Yaskawa INFORM job: X2_102(P)(90,-90)1.JBI

/JOB
//NAME X2_102(P)(90,-90)1
//POS
///NPOS 230,230,226,13,0,0
///TOOL 0
///POSTYPE PULSE
///PULSE
C00000=2000,-138093,-117084,0,0,0
C00001=4305,236497,208118,-17761,33698,0
C00002=-59706,236497,171970,-17761,33698,0
C00003=-68642,233553,162335,18407,63943,-60167
C00004=-68620,237873,184689,20710,53031,-62187
C00005=-67493,232083,179997,20020,52672,-61765
C00006=-67050,229604,177876,19730,52595,-61585
C00007=-67044,229502,178985,19916,51901,-61724
C00008=-67038,229450,178497,19841,52157,-61669
C00009=-66578,226776,174924,19337,52827,-61332
C00010=-67038,229450,178497,19841,52157,-61669
C00011=-68631,234094,163892,18504,63294,-60271
C00012=-68145,241811,194493,16574,45015,-61509
C00013=-67317,229778,184749,15987,44670,-61166
C00014=-67317,229387,185455,16165,44058,-61279
C00015=-67317,229778,184749,15987,44670,-61166
C00016=-66834,227293,181425,15407,45318,-60815
C00017=-67317,229778,184749,15987,44670,-61166
C00018=-68701,238087,188501,16512,46831,-61441
C00019=-66679,248207,214141,19957,35663,-62952
C00020=-66362,236944,211229,20590,32234,-63605
C00021=-65277,231220,208227,19566,31083,-63125
C00022=-65277,230538,208245,19768,30741,-63230
C00023=-65277,231220,208227,19566,31083,-63125
C00024=-64770,229332,205657,18720,31545,-62649
C00025=-65277,231220,208227,19566,31083,-63125
C00026=-63899,247748,213566,15829,35762,-61053
C00027=-132961,256009,219351,-662,67771,16322
C00028=-150721,258133,220838,-4903,56597,36219
C00029=-175956,234235,210676,-21015,30395,63926
C00030=-177622,226369,202159,-18586,31129,62559
C00031=-177622,225563,202167,-18810,30730,62676
C00032=-177622,225876,202166,-18723,30883,62631
C00033=-178207,223412,198783,-17689,31531,62057
C00034=-177236,228737,204255,-19030,31146,62814
C00035=-175884,240118,209836,-19152,33747,62947
C00036=-173679,229857,186287,-16925,43983,61731
C00037=-173679,227981,188546,-17672,41731,62191
C00038=-173679,227243,189165,-17934,41006,62348
C00039=-173679,227551,188921,-17828,41299,62281
C00040=-174254,224827,185246,-17073,41999,61834
C00041=-173679,227551,188921,-17828,41299,62281
C00042=-173139,236491,197187,-18441,40951,62645
C00043=-172603,232602,161257,-18712,64089,60261
C00044=-173924,235628,180815,-18889,51873,61342
C00045=-172608,237232,184033,-21073,53108,62337
C00046=-173740,231415,179286,-20377,52761,61910
C00047=-174186,228920,177136,-20083,52691,61728
C00048=-174192,228817,178244,-20271,51998,61869
C00049=-174189,228638,177277,-20141,52472,61772
C00050=-174651,225918,173635,-19633,53157,61430
C00051=-174189,228638,177277,-20141,52472,61772
C00052=-172611,236980,184222,-21136,52878,62385
C00053=-172606,232705,161920,-18764,63751,60317
C00054=-33909,232602,161257,-18712,64089,60261
C00055=-15700,2243,-58558,-65367,94407,-58645
C00056=-42038,-24148,-64629,-54323,75559,-58717
C00057=-44197,-22959,-60659,-53735,73332,-58425
C00058=-45039,-22397,-59015,-53526,72451,-58312
C00059=-44979,-23271,-57928,-53825,71802,-57871
C00060=-44992,-23122,-58143,-53767,71922,-57954
C00061=-46191,-21439,-56856,-53216,71335,-58219
C00062=-44992,-23122,-58143,-53767,71922,-57954
C00063=-41989,-25009,-63827,-54529,75024,-58350
C00064=-32524,-34812,-71854,-58522,80038,-56653
C00065=-45017,-81581,-97017,-55472,68259,-55558
C00066=-56084,-63511,-88405,-49217,64831,-59493
C00067=-58462,-60349,-83704,-48479,62782,-59568
C00068=-59376,-59036,-81788,-48205,61981,-59596
C00069=-59311,-59777,-80503,-48699,61221,-59131
C00070=-59003,-60257,-81034,-48822,61431,-59087
C00071=-60302,-57702,-79583,-47994,61058,-59566
C00072=-59003,-60257,-81034,-48822,61431,-59087
C00073=-55681,-64881,-87691,-49815,64278,-58966
C00074=-45017,-81581,-97017,-55472,68259,-55558
C00075=-32894,-34432,-71630,-58366,79867,-56737
C00076=-41688,-24576,-64954,-54484,75728,-58645
C00077=-43859,-23403,-60999,-53891,73497,-58353
C00078=-44706,-22847,-59360,-53679,72615,-58240
C00079=-44645,-23721,-58271,-53976,71967,-57798
C00080=-44682,-23582,-58448,-53916,72056,-57875
C00081=-45888,-21907,-57169,-53364,71466,-58140
C00082=-44682,-23582,-58448,-53916,72056,-57875
C00083=-41663,-25454,-64115,-54683,75164,-58270
C00084=-32894,-34432,-71630,-58366,79867,-56737
C00085=-30502,-36607,-73062,-59339,81056,-56251
C00086=-41630,-24614,-65007,-54508,75766,-58639
C00087=-43802,-23446,-61055,-53913,73534,-58347
C00088=-44650,-22892,-59418,-53701,72651,-58234
C00089=-44589,-23766,-58329,-53998,72004,-57792
C00090=-44608,-23720,-58520,-53955,72080,-57850
C00091=-45815,-22046,-57244,-53403,71488,-58116
C00092=-44608,-23720,-58520,-53955,72080,-57850
C00093=-41584,-25591,-64184,-54723,75189,-58245
C00094=-30502,-36607,-73062,-59339,81056,-56251
C00095=-30521,-36804,-72907,-59354,80942,-56176
C00096=-41810,-24598,-64713,-54460,75569,-58606
C00097=-43977,-23401,-60743,-53873,73340,-58316
C00098=-44823,-22836,-59099,-53664,72459,-58203
C00099=-44777,-23490,-58282,-53888,71973,-57872
C00100=-44767,-23386,-58412,-53859,72059,-57922
C00101=-45672,-22131,-57454,-53445,71616,-58121
C00102=-44767,-23386,-58412,-53859,72059,-57922
C00103=-41752,-25252,-64079,-54627,75166,-58318
C00104=-30521,-36804,-72907,-59354,80942,-56176
C00105=-48617,-100899,-104901,-55908,63245,-54221
C00106=-60981,-78178,-95502,-47940,60221,-59456
C00107=-63421,-73970,-90529,-47045,58377,-59730
C00108=-64353,-72276,-88515,-46711,57655,-59831
C00109=-64286,-72889,-87139,-47282,56881,-59359
C00110=-64274,-72850,-87331,-47224,56982,-59410
C00111=-65583,-69919,-85834,-46243,56736,-59988
C00112=-64274,-72850,-87331,-47224,56982,-59410
C00113=-57432,-98051,-106862,-51065,59935,-57313
C00114=-51188,-107076,-112538,-52509,60337,-56355
C00115=-83162,-143293,-113239,4095,19388,-67719
C00116=-87059,-126422,-104497,10100,20417,-69023
C00117=-85148,-116277,-98792,5838,21915,-66988
C00118=-84341,-113269,-97174,4239,22413,-66225
C00119=-41354,-51421,-69594,-68729,84300,-42170
C00120=-66411,-100108,-97884,-57632,66468,-44476
C00121=-56302,-60377,-70344,-75389,89529,-53167
C00122=-54473,-59290,-70505,-75710,90966,-53293
C00123=-50946,-58104,-72389,-76445,93850,-53772
C00124=-34731,-98541,-90949,-75868,93293,-49305
C00125=-38562,-61143,-74059,-78354,102200,-52510
C00126=-51313,-57535,-72089,-76390,93628,-53853
C00127=-54828,-58696,-70195,-75657,90754,-53377
C00128=-56440,-59997,-70035,-75367,89439,-53183
C00129=-93781,-139674,-106819,-38352,21241,-56382
C00130=-61530,-99076,-95664,-44966,45788,-52630
C00131=-83648,-111417,-96267,2924,22775,-65596
C00132=-85460,-115209,-98453,6324,22277,-67219
C00133=-87376,-128198,-110756,9444,23354,-68706
C00134=-66110,-162513,-113557,-65322,17781,-32754
C00135=-60362,-179762,-121914,-78103,19027,-26385
C00136=-78271,-141405,-108666,-10042,15201,-59438
C00137=-76792,-129799,-102924,-12030,17790,-58472
C00138=-74738,-129134,-99045,-25052,13652,-53297
C00139=-36188,-62041,-77688,-66032,84757,-42278
C00140=-46102,-88609,-90371,-65502,79628,-40662
C00141=-43207,-58645,-71334,-74593,95184,-49845
C00142=-41791,-47729,-64018,-78026,100149,-53095
C00143=-38644,-45375,-65147,-79031,102736,-53739
C00144=-22542,-58930,-72906,-80701,113358,-51531
C00145=-45507,-85827,-81768,-80030,94289,-48289
C00146=-21007,-49469,-63567,-84664,112915,-50403
C00147=-24143,-52779,-63157,-83372,110435,-49576
C00148=-25588,-55109,-63516,-82813,109262,-49172
C00149=-29213,-141193,-106326,-70590,66679,-33929
C00150=-21677,-102038,-94363,-66600,73853,-38839
C00151=-30241,-129324,-100953,-69122,50791,-33041
C00152=-46232,-152372,-104130,-83256,26044,-24905
C00153=-44377,-165065,-109179,-90053,27028,-21315
C00154=-311,-178979,-111450,-86459,56764,-16230
C00155=-59708,-176831,-116235,-83669,15342,-24345
C00156=-79056,-141883,-108790,-8064,14946,-60379
C00157=-77513,-130262,-103056,-10505,17536,-59201
C00158=-74170,-126151,-101228,-19436,19691,-55187
C00159=-36840,-62408,-78088,-65333,83828,-45019
C00160=-50437,-100078,-97430,-60201,71072,-46441
C00161=-45392,-83282,-85893,-68940,82387,-50193
C00162=-37649,-79344,-88446,-70118,88865,-50776
C00163=-26650,-88423,-96706,-71980,96311,-49687
C00164=-27360,-157090,-119697,-70425,73735,-40403
C00165=-26933,-67218,-77205,-79449,109983,-51051
C00166=-40780,-54413,-70384,-78301,100955,-53239
C00167=-44144,-56530,-69031,-77374,98185,-52627
C00168=-46739,-82554,-83925,-71442,84833,-50278
C00169=-64576,-133797,-108987,-56957,49971,-40299
C00170=-55730,-116486,-104453,-54149,57147,-39702
C00171=-64775,-126412,-104837,-43035,33616,-45207
C00172=-84360,-137825,-105111,6410,14710,-67243
C00173=-83782,-174049,-119465,14191,4988,-70704
C00174=4306,-189564,-118248,-76797,69073,-14089
C00175=-9355,229277,174760,14349,4120,-60080
C00176=-63851,249906,184838,11388,54090,-58270
C00177=-66966,229251,175893,14496,49590,-60184
C00178=-66966,228979,178450,14872,47930,-60442
C00179=-66981,229181,177726,14757,48464,-60364
C00180=-67823,233206,185230,16003,46159,-61141
C00181=-66981,228894,179384,15025,47334,-60544
C00182=-66990,228821,179287,15027,47357,-60545
C00183=-66967,228791,179403,15048,47276,-60547
C00184=-66961,228789,179266,15001,47362,-60537
C00185=-66965,228460,180628,15248,46388,-60700
C00186=-66802,227674,179068,14990,46895,-60538
C00187=-66779,227397,179466,15054,46528,-60590
C00188=-66807,226773,182027,15552,44699,-60914
C00189=-66832,224442,185298,16520,41608,-61494
C00190=-66840,224422,185215,16494,41648,-61489
C00191=-66820,223938,186111,16728,40875,-61637
C00192=-66853,222022,186802,17225,39537,-61929
C00193=-66912,216121,188235,18844,35797,-62842
C00194=-66885,216347,188464,18827,35771,-62831
C00195=-66952,215633,187924,18914,35747,-62874
C00196=-67008,215777,188020,18974,35761,-62903
C00197=-64896,228147,204946,18938,31412,-62768
C00198=-64451,229383,207615,19004,30362,-62779
C00199=-64319,229986,208437,18975,30146,-62755
C00200=-64320,235654,207860,17333,33259,-61891
C00201=-127852,233528,172858,-1116,53739,8677
C00202=-174263,228432,175140,-14901,49789,60445
C00203=-174268,228211,177769,-15284,48114,60710
C00204=-174246,228391,177829,-15287,48171,60710
C00205=-173475,232193,184234,-16357,46404,61376
C00206=-174246,228181,178891,-15468,47435,60832
C00207=-174240,228133,178826,-15469,47451,60832
C00208=-174271,228016,178845,-15463,47379,60831
C00209=-174276,227918,178508,-15413,47528,60799
C00210=-174286,227658,179844,-15655,46590,60950
C00211=-174351,227295,179377,-15579,46676,60907
C00212=-174332,227272,179929,-15676,46343,60972
C00213=-174371,226155,181833,-16121,44653,61258
C00214=-174192,224903,185875,-17238,41679,61934
C00215=-174186,224802,185663,-17218,41757,61925
C00216=-174205,224201,186288,-17427,41100,62055
C00217=-174226,222498,187148,-17913,39751,62341
C00218=-174338,216137,187971,-19375,36146,63177
C00219=-174344,216285,188030,-19351,36181,63161
C00220=-174327,216170,187871,-19349,36222,63161
C00221=-174333,215937,187942,-19432,36065,63204
C00222=-174325,215982,187948,-19443,36091,63210
C00223=-176900,230407,207583,-19326,31072,63020
C00224=-176902,229512,207806,-19651,30509,63187
C00225=-177018,230048,208538,-19629,30316,63168
C00226=-177017,235510,208022,-18011,33280,62316
C00227=-177018,208627,156143,-19629,29463,63168
C00228=4305,194232,136177,-17761,33698,62179
C00229=2000,-138093,-117084,0,0,0
BC00000=166720,666220,1057063
BC00001=32490,666220,1075175
BC00002=32490,666220,1075175
BC00003=108321,818406,1075175
BC00004=108321,818406,1075175
BC00005=108321,818406,1075175
BC00006=108321,818406,1075175
BC00007=108321,818406,1075175
BC00008=108321,818406,1075175
BC00009=108321,818406,1075175
BC00010=108321,818406,1075175
BC00011=108321,818406,1075175
BC00012=112515,736490,1075175
BC00013=112515,736490,1075175
BC00014=112515,736490,1075175
BC00015=112515,736490,1075175
BC00016=112515,736490,1075175
BC00017=112515,736490,1075175
BC00018=112515,736490,1075175
BC00019=112881,691782,1025034
BC00020=113047,671527,1002318
BC00021=113089,666372,996537
BC00022=113089,666372,996537
BC00023=113089,666372,996537
BC00024=113089,666372,996537
BC00025=113089,666372,996537
BC00026=113089,666372,996537
BC00027=249276,665500,992981
BC00028=284297,665276,992066
BC00029=334133,666220,990764
BC00030=334133,666220,990764
BC00031=334133,666220,990764
BC00032=334133,666220,990764
BC00033=334133,666220,990764
BC00034=334133,666220,990764
BC00035=334133,666220,990764
BC00036=325487,705237,1075175
BC00037=325487,705237,1075175
BC00038=325487,705237,1075175
BC00039=325487,705237,1075175
BC00040=325487,705237,1075175
BC00041=325487,705237,1075175
BC00042=325487,705237,1075175
BC00043=330094,817929,1075175
BC00044=331720,756851,1041191
BC00045=330094,817929,1075175
BC00046=330094,817929,1075175
BC00047=330094,817929,1075175
BC00048=330094,817929,1075175
BC00049=330094,817929,1075175
BC00050=330094,817929,1075175
BC00051=330094,817929,1075175
BC00052=330094,817929,1075175
BC00053=330094,817929,1075175
BC00054=52198,668359,1075175
BC00055=166720,666220,1057063
BC00056=216765,666220,1057063
BC00057=216765,666220,1057063
BC00058=216765,666220,1057063
BC00059=216765,666220,1057063
BC00060=216765,666220,1057063
BC00061=216765,666220,1057063
BC00062=216765,666220,1057063
BC00063=216765,666220,1057063
BC00064=216765,666220,1057063
BC00065=189956,666220,1056793
BC00066=189956,666220,1056793
BC00067=189956,666220,1056793
BC00068=189956,666220,1056793
BC00069=189956,666220,1056793
BC00070=189956,666220,1056793
BC00071=189956,666220,1056793
BC00072=189956,666220,1056793
BC00073=189956,666220,1056793
BC00074=189956,666220,1056793
BC00075=95589,666220,1056895
BC00076=95589,666220,1056895
BC00077=95589,666220,1056895
BC00078=95589,666220,1056895
BC00079=95589,666220,1056895
BC00080=95589,666220,1056895
BC00081=95589,666220,1056895
BC00082=95589,666220,1056895
BC00083=95589,666220,1056895
BC00084=95589,666220,1056895
BC00085=65057,666220,1056713
BC00086=65057,666220,1056713
BC00087=65057,666220,1056713
BC00088=65057,666220,1056713
BC00089=65057,666220,1056713
BC00090=65057,666220,1056713
BC00091=65057,666220,1056713
BC00092=65057,666220,1056713
BC00093=65057,666220,1056713
BC00094=65057,666220,1056713
BC00095=13150,666220,1055634
BC00096=13150,666220,1055634
BC00097=13150,666220,1055634
BC00098=13150,666220,1055634
BC00099=13150,666220,1055634
BC00100=13150,666220,1055634
BC00101=13150,666220,1055634
BC00102=13150,666220,1055634
BC00103=13150,666220,1055634
BC00104=13150,666220,1055634
BC00105=15,666220,1056645
BC00106=15,666220,1056645
BC00107=15,666220,1056645
BC00108=15,666220,1056645
BC00109=15,666220,1056645
BC00110=15,666220,1056645
BC00111=15,666220,1056645
BC00112=15,666220,1056645
BC00113=15,666220,1056645
BC00114=15,666220,1056645
BC00115=23745,686641,1073486
BC00116=26125,688689,1075175
BC00117=26125,688689,1075175
BC00118=26125,688689,1075175
BC00119=26125,688689,1075175
BC00120=26125,688689,1075175
BC00121=26125,688689,1075175
BC00122=26125,688689,1075175
BC00123=26125,688689,1075175
BC00124=26125,688689,1075175
BC00125=284154,689569,1075175
BC00126=284154,689569,1075175
BC00127=284154,689569,1075175
BC00128=284154,689569,1075175
BC00129=284154,689569,1075175
BC00130=284154,689569,1075175
BC00131=284154,689569,1075175
BC00132=284154,689569,1075175
BC00133=284154,689569,1075175
BC00134=284154,689569,1075175
BC00135=166821,701812,1075175
BC00136=166821,701812,1075175
BC00137=166821,701812,1075175
BC00138=166821,701812,1075175
BC00139=166821,701812,1075175
BC00140=166821,701812,1075175
BC00141=166821,701812,1075174
BC00142=166821,701812,1075175
BC00143=166821,701812,1075175
BC00144=166821,701812,1075175
BC00145=107577,675403,1075175
BC00146=60976,728964,1075175
BC00147=60976,728964,1075175
BC00148=60976,728964,1075175
BC00149=60976,728964,1075175
BC00150=60976,728964,1075175
BC00151=60975,728964,1075174
BC00152=60976,728964,1075175
BC00153=60976,728964,1075175
BC00154=60976,728964,1075175
BC00155=214157,701974,1075175
BC00156=214157,701974,1075175
BC00157=214157,701974,1075175
BC00158=214157,701974,1075175
BC00159=214157,701974,1075175
BC00160=214157,701974,1075175
BC00161=214157,701974,1075175
BC00162=214157,701974,1075175
BC00163=214157,701974,1075175
BC00164=214157,701974,1075175
BC00165=126731,702207,1075175
BC00166=126731,702207,1075175
BC00167=126731,702207,1075175
BC00168=126731,702207,1075175
BC00169=126731,702207,1075175
BC00170=126731,702207,1075175
BC00171=126731,702207,1075175
BC00172=126731,702207,1075175
BC00173=126731,702207,1075175
BC00174=126731,702207,1075175
BC00175=0,671300,1075175
BC00176=102033,814443,1075175
BC00177=104277,804739,1075175
BC00178=109889,805427,1075175
BC00179=112133,805702,1075175
BC00180=112133,805702,1075175
BC00181=112133,805702,1075175
BC00182=112133,805702,1075175
BC00183=112115,811337,1075171
BC00184=112235,790267,1075175
BC00185=112385,757219,1075175
BC00186=112368,762877,1075175
BC00187=112401,759711,1075175
BC00188=112515,736490,1075175
BC00189=112651,705808,1075172
BC00190=112632,711465,1075175
BC00191=112664,708917,1075175
BC00192=112731,698583,1075175
BC00193=112912,671578,1075175
BC00194=112897,675330,1075175
BC00195=112903,675530,1064805
BC00196=112969,667577,1038313
BC00197=113089,666372,996537
BC00198=110434,666220,999205
BC00199=104822,666220,1018123
BC00200=104780,666220,1075175
BC00201=236932,745843,1075175
BC00202=332819,804241,1075175
BC00203=327209,804894,1075175
BC00204=324965,805156,1075175
BC00205=324965,805156,1075175
BC00206=324965,805156,1075175
BC00207=324965,805156,1075175
BC00208=324947,810790,1075175
BC00209=325043,789742,1075175
BC00210=325218,756702,1075175
BC00211=325200,762360,1075175
BC00212=325209,759192,1075175
BC00213=325324,735955,1075175
BC00214=325487,705242,1075175
BC00215=325468,710849,1075175
BC00216=325473,708338,1075175
BC00217=325540,697985,1075175
BC00218=325697,671186,1075175
BC00219=325677,676538,1075175
BC00220=325677,676538,1075175
BC00221=325711,674865,1062596
BC00222=325783,666243,1034429
BC00223=325896,666237,989644
BC00224=328141,666220,997078
BC00225=333753,666220,1016016
BC00226=333712,666220,1075175
BC00227=333753,666220,1016016
BC00228=32490,666220,1075175
BC00229=166720,666220,1057063
EC00000=798156,-556475
EC00001=798156,-556920
EC00002=798156,-556920
EC00003=443420,-556475
EC00004=443420,-556475
EC00005=443420,-556475
EC00006=443420,-556475
EC00007=443420,-556475
EC00008=443420,-556475
EC00009=443420,-556475
EC00010=443420,-556475
EC00011=443420,-556475
EC00012=657016,-556187
EC00013=657016,-556187
EC00014=657016,-556187
EC00015=657016,-556187
EC00016=657016,-556187
EC00017=657016,-556187
EC00018=657016,-556187
EC00019=846901,-556371
EC00020=932929,-556454
EC00021=954822,-556475
EC00022=954822,-556475
EC00023=954822,-556475
EC00024=954822,-556475
EC00025=954822,-556475
EC00026=954822,-556475
EC00027=958275,-556749
EC00028=959163,-556820
EC00029=960426,-556920
EC00030=960426,-556920
EC00031=960426,-556920
EC00032=960426,-556920
EC00033=960426,-556920
EC00034=960426,-556920
EC00035=960426,-556920
EC00036=736908,-556362
EC00037=736908,-556362
EC00038=736908,-556362
EC00039=736908,-556362
EC00040=736908,-556362
EC00041=736908,-556362
EC00042=736908,-556362
EC00043=443420,-556475
EC00044=651568,-556654
EC00045=443420,-556475
EC00046=443420,-556475
EC00047=443420,-556475
EC00048=443420,-556475
EC00049=443420,-556475
EC00050=443420,-556475
EC00051=443420,-556475
EC00052=443420,-556475
EC00053=443420,-556475
EC00054=663289,-556475
EC00055=798156,-556475
EC00056=798156,-556475
EC00057=798156,-556475
EC00058=798156,-556475
EC00059=798156,-556475
EC00060=798156,-556475
EC00061=798156,-556475
EC00062=798156,-556475
EC00063=798156,-556475
EC00064=798156,-556475
EC00065=798156,-556475
EC00066=798156,-556475
EC00067=798156,-556475
EC00068=798156,-556475
EC00069=798156,-556475
EC00070=798156,-556475
EC00071=798156,-556475
EC00072=798156,-556475
EC00073=798156,-556475
EC00074=798156,-556475
EC00075=798156,-556475
EC00076=798156,-556475
EC00077=798156,-556475
EC00078=798156,-556475
EC00079=798156,-556475
EC00080=798156,-556475
EC00081=798156,-556475
EC00082=798156,-556475
EC00083=798156,-556475
EC00084=798156,-556475
EC00085=798156,-556475
EC00086=798156,-556475
EC00087=798156,-556475
EC00088=798156,-556475
EC00089=798156,-556475
EC00090=798156,-556475
EC00091=798156,-556475
EC00092=798156,-556475
EC00093=798156,-556475
EC00094=798156,-556475
EC00095=798156,-556475
EC00096=798156,-556475
EC00097=798156,-556475
EC00098=798156,-556475
EC00099=798156,-556475
EC00100=798156,-556475
EC00101=798156,-556475
EC00102=798156,-556475
EC00103=798156,-556475
EC00104=798156,-556475
EC00105=798156,-556475
EC00106=798156,-556475
EC00107=798156,-556475
EC00108=798156,-556475
EC00109=798156,-556475
EC00110=798156,-556475
EC00111=798156,-556475
EC00112=798156,-556475
EC00113=798156,-556475
EC00114=798156,-556475
EC00115=798156,-556475
EC00116=798156,-556475
EC00117=798156,-556475
EC00118=798156,-556475
EC00119=798156,-556475
EC00120=798156,-556475
EC00121=798156,-556475
EC00122=798156,-556475
EC00123=798156,-556475
EC00124=798156,-556475
EC00125=798156,-556475
EC00126=798156,-556475
EC00127=798156,-556475
EC00128=798156,-556475
EC00129=798156,-556475
EC00130=798156,-556475
EC00131=798156,-556475
EC00132=798156,-556475
EC00133=798156,-556475
EC00134=798156,-556475
EC00135=798156,-556475
EC00136=798156,-556475
EC00137=798156,-556475
EC00138=798156,-556475
EC00139=798156,-556475
EC00140=798156,-556475
EC00141=798155,-556475
EC00142=798156,-556475
EC00143=798156,-556475
EC00144=798156,-556475
EC00145=798156,-556475
EC00146=798156,-556475
EC00147=798156,-556475
EC00148=798156,-556475
EC00149=798156,-556475
EC00150=798156,-556475
EC00151=798155,-556475
EC00152=798156,-556475
EC00153=798156,-556475
EC00154=798156,-556475
EC00155=798156,-556475
EC00156=798156,-556475
EC00157=798156,-556475
EC00158=798156,-556475
EC00159=798156,-556475
EC00160=798156,-556475
EC00161=798156,-556475
EC00162=798156,-556475
EC00163=798156,-556475
EC00164=798156,-556475
EC00165=798156,-556475
EC00166=798156,-556475
EC00167=798156,-556475
EC00168=798156,-556475
EC00169=798156,-556475
EC00170=798156,-556475
EC00171=798156,-556475
EC00172=798156,-556475
EC00173=798156,-556475
EC00174=798156,-556475
EC00175=798156,-556475
EC00176=449706,-555609
EC00177=449706,-555609
EC00178=449706,-555609
EC00179=449706,-555609
EC00180=449706,-555609
EC00181=449704,-555609
EC00182=497563,-555770
EC00183=577410,-555996
EC00184=577410,-555996
EC00185=593464,-556037
EC00186=657016,-556187
EC00187=736906,-556362
EC00188=736908,-556362
EC00189=752993,-556395
EC00190=784818,-556475
EC00191=864675,-556475
EC00192=864752,-556475
EC00193=880165,-556475
EC00194=910304,-556475
EC00195=954822,-556475
EC00196=960426,-556475
EC00197=960426,-556475
EC00198=960426,-556475
EC00199=665239,-555975
EC00200=449706,-555609
EC00201=449706,-555609
EC00202=449706,-555609
EC00203=449706,-555609
EC00204=449706,-555609
EC00205=497563,-555770
EC00206=577410,-555996
EC00207=577410,-555996
EC00208=593464,-556037
EC00209=657016,-556187
EC00210=736908,-556362
EC00211=736908,-556362
EC00212=752993,-556395
EC00213=784818,-556475
EC00214=863892,-556660
EC00215=864791,-556662
EC00216=864791,-556662
EC00217=880786,-556704
EC00218=912696,-556789
EC00219=960272,-556920
EC00220=960426,-556920
EC00221=960426,-556920
EC00222=960426,-556920
EC00223=960426,-556920
EC00224=960426,-556920
EC00225=798156,-556475
///POSTYPE BASE
///RECTAN
///RCONF 0,0,0,0,0,0,0,0,0,0,0,0,0,0,0,0,0,0,0,0,0,0,0,0
P00006=0.222,-3.123,-1.508,0.0000,0.0000,0.0000
P00021=-0.225,-6.128,-0.405,0.0000,0.0000,0.0000
P00022=0.222,-3.123,-1.508,0.0000,0.0000,0.0000
P00023=0.143,-0.036,0.682,0.0000,0.0000,0.0000
P00024=0.145,-0.552,1.326,0.0000,0.0000,0.0000
P00025=-2.003,0.006,0.728,0.0000,0.0000,0.0000
P00026=0.562,-0.002,-0.337,0.0000,0.0000,0.0000
P00027=-0.746,0.015,-9.096,0.0000,0.0000,0.0000
P00028=-2.237,-0.018,-7.702,0.0000,0.0000,0.0000
P00066=5.557,-0.028,3.115,0.0000,0.0000,0.0000
///RCONF 0,1,0,0,0,0,0,0,0,0,0,0,0,0,0,0,0,0,0,0,0,0,0,0
P00067=-0.081,0.026,-1.119,0.0000,0.0000,0.0000
///RCONF 0,0,0,0,0,0,0,0,0,0,0,0,0,0,0,0,0,0,0,0,0,0,0,0
P00068=2.896,1.192,4.622,0.0000,0.0000,0.0000
///RCONF 0,1,0,0,0,0,0,0,0,0,0,0,0,0,0,0,0,0,0,0,0,0,0,0
P00075=-1.802,0.025,1.546,0.0000,0.0000,0.0000
//INST
///DATE 2024/04/10 12:22
///ATTR SC,RW
///GROUP1 RB1,BS1
///GROUP2 ST1
NOP
'X2_102(P)(90,-90)1
MOVJ C00000 BC00000 VJ=100.00  +MOVJ EC00000 VJ=100.00
MOVJ C00001 BC00001 VJ=100.00  +MOVJ EC00001 VJ=100.00
MOVJ C00002 BC00002 VJ=100.00  +MOVJ EC00002 VJ=100.00
'Path S3368
SFTOF3D
MOVJ C00003 BC00003 VJ=100.00  +MOVJ EC00003 VJ=100.00
MOVJ C00004 BC00004 VJ=100.00  +MOVJ EC00004 VJ=100.00
MOVL C00005 BC00005 V=800.0  +MOVJ EC00005 VJ=100.00
SMOVL C00006 BC00006 V=166.7  +MOVJ EC00006
SREFP 3 C00007 BC00007  +REFP EC00007
CALL JOB:SEARCH-R1-S13D
SET P027 P006
SFTON3D P027
SMOVL C00008 BC00008 V=166.7  +MOVJ EC00008
SREFP 3 C00009 BC00009  +REFP EC00009
CALL JOB:SEARCH-R1-S13D
SET P027 P006
SFTON3D P027
SMOVL C00010 BC00010 V=166.7  +MOVJ EC00010
MOVL C00011 BC00011 V=1000.0  +MOVJ EC00011 VJ=100.00
'EndPath S3368
'Path S3369
SFTOF3D
MOVJ C00012 BC00012 VJ=100.00  +MOVJ EC00012 VJ=100.00
SMOVL C00013 BC00013 V=250.0  +MOVJ EC00013
SREFP 3 C00014 BC00014  +REFP EC00014
CALL JOB:SEARCH-R1-S13D
SET P066 P006
SFTON3D P066
SMOVL C00015 BC00015 V=166.7  +MOVJ EC00015
SREFP 3 C00016 BC00016  +REFP EC00016
CALL JOB:SEARCH-R1-S13D
SET P066 P006
SFTON3D P066
SMOVL C00017 BC00017 V=250.0  +MOVJ EC00017
SFTOF3D
MOVJ C00018 BC00018 VJ=100.00  +MOVJ EC00018 VJ=100.00
MOVJ C00019 BC00019 VJ=100.00  +MOVJ EC00019 VJ=100.00
MOVJ C00020 BC00020 VJ=100.00  +MOVJ EC00020 VJ=100.00
SMOVL C00021 BC00021 V=250.0  +MOVJ EC00021
SREFP 3 C00022 BC00022  +REFP EC00022
CALL JOB:SEARCH-R1-S13D
SET P067 P006
SFTON3D P067
SMOVL C00023 BC00023 V=166.7  +MOVJ EC00023
SREFP 3 C00024 BC00024  +REFP EC00024
CALL JOB:SEARCH-R1-S13D
SET P067 P006
SFTON3D P067
SMOVL C00025 BC00025 V=250.0  +MOVJ EC00025
SFTOF3D
MOVJ C00026 BC00026 VJ=100.00  +MOVJ EC00026 VJ=100.00
MOVJ C00027 BC00027 VJ=40.00  +MOVJ EC00027 VJ=100.00
MOVJ C00028 BC00028 VJ=80.00  +MOVJ EC00028 VJ=100.00
SFTOF3D
MOVJ C00029 BC00029 VJ=80.00  +MOVJ EC00029 VJ=100.00
SMOVL C00030 BC00030 V=166.7  +MOVJ EC00030
SREFP 3 C00031 BC00031  +REFP EC00031
CALL JOB:SEARCH-R1-S13D
SET P068 P006
SFTON3D P068
SMOVL C00032 BC00032 V=166.7  +MOVJ EC00032
SREFP 3 C00033 BC00033  +REFP EC00033
CALL JOB:SEARCH-R1-S13D
SET P068 P006
SFTON3D P068
SMOVL C00034 BC00034 V=250.0  +MOVJ EC00034
SFTOF3D
MOVJ C00035 BC00035 VJ=80.00  +MOVJ EC00035 VJ=80.00
MOVJ C00036 BC00036 VJ=100.00  +MOVJ EC00036 VJ=100.00
SFTOF3D
SMOVL C00037 BC00037 V=166.7  +MOVJ EC00037
SREFP 3 C00038 BC00038  +REFP EC00038
CALL JOB:SEARCH-R1-S13D
SET P075 P006
SFTON3D P075
SMOVL C00039 BC00039 V=166.7  +MOVJ EC00039
SREFP 3 C00040 BC00040  +REFP EC00040
CALL JOB:SEARCH-R1-S13D
SET P075 P006
SFTON3D P075
SMOVL C00041 BC00041 V=250.0  +MOVJ EC00041
SFTOF3D
MOVL C00042 BC00042 V=1000.0  +MOVJ EC00042 VJ=100.00
MOVJ C00043 BC00043 VJ=100.00  +MOVJ EC00043 VJ=100.00
MOVJ C00044 BC00044 VJ=100.00  +MOVJ EC00044 VJ=100.00
MOVJ C00045 BC00045 VJ=100.00  +MOVJ EC00045 VJ=100.00
MOVL C00046 BC00046 V=800.0  +MOVJ EC00046 VJ=100.00
SMOVL C00047 BC00047 V=166.7  +MOVJ EC00047
SREFP 3 C00048 BC00048  +REFP EC00048
CALL JOB:SEARCH-R1-S13D
SET P028 P006
SFTON3D P028
SMOVL C00049 BC00049 V=166.7  +MOVJ EC00049
SREFP 3 C00050 BC00050  +REFP EC00050
CALL JOB:SEARCH-R1-S13D
SET P028 P006
SFTON3D P028
SMOVL C00051 BC00051 V=250.0  +MOVJ EC00051
MOVL C00052 BC00052 V=1000.0  +MOVJ EC00052 VJ=100.00
MOVL C00053 BC00053 V=1000.0  +MOVJ EC00053 VJ=100.00
'EndPath S3369
MOVJ C00054 BC00054 VJ=100.00  +MOVJ EC00054 VJ=100.00
'
MOVJ C00055 BC00055 VJ=100.00  +MOVJ EC00055 VJ=100.00
'Path S3399
SFTOF3D
MOVJ C00056 BC00056 VJ=100.00  +MOVJ EC00056 VJ=100.00
MOVL C00057 BC00057 V=800.0  +MOVJ EC00057 VJ=100.00
SMOVL C00058 BC00058 V=166.7  +MOVJ EC00058
SREFP 3 C00059 BC00059  +REFP EC00059
CALL JOB:SEARCH-R1-S13D
SET P021 P006
SFTON3D P021
SMOVL C00060 BC00060 V=166.7  +MOVJ EC00060
SREFP 3 C00061 BC00061  +REFP EC00061
CALL JOB:SEARCH-R1-S13D
SET P021 P006
SFTON3D P021
SMOVL C00062 BC00062 V=166.7  +MOVJ EC00062
MOVL C00063 BC00063 V=1000.0  +MOVJ EC00063 VJ=100.00
'EndPath S3399
MOVJ C00064 BC00064 VJ=100.00  +MOVJ EC00064 VJ=100.00
MOVJ C00065 BC00065 VJ=100.00  +MOVJ EC00065 VJ=100.00
'Path S3400
SFTOF3D
MOVJ C00066 BC00066 VJ=100.00  +MOVJ EC00066 VJ=100.00
MOVL C00067 BC00067 V=800.0  +MOVJ EC00067 VJ=100.00
SMOVL C00068 BC00068 V=166.7  +MOVJ EC00068
SREFP 3 C00069 BC00069  +REFP EC00069
CALL JOB:SEARCH-R1-S13D
SET P022 P006
SFTON3D P022
SMOVL C00070 BC00070 V=166.7  +MOVJ EC00070
SREFP 3 C00071 BC00071  +REFP EC00071
CALL JOB:SEARCH-R1-S13D
SET P022 P006
SFTON3D P022
SMOVL C00072 BC00072 V=166.7  +MOVJ EC00072
MOVL C00073 BC00073 V=1000.0  +MOVJ EC00073 VJ=100.00
'EndPath S3400
MOVJ C00074 BC00074 VJ=100.00  +MOVJ EC00074 VJ=100.00
MOVJ C00075 BC00075 VJ=100.00  +MOVJ EC00075 VJ=100.00
'Path S3401
SFTOF3D
MOVJ C00076 BC00076 VJ=100.00  +MOVJ EC00076 VJ=100.00
MOVL C00077 BC00077 V=800.0  +MOVJ EC00077 VJ=100.00
SMOVL C00078 BC00078 V=166.7  +MOVJ EC00078
SREFP 3 C00079 BC00079  +REFP EC00079
CALL JOB:SEARCH-R1-S13D
SET P023 P006
SFTON3D P023
SMOVL C00080 BC00080 V=166.7  +MOVJ EC00080
SREFP 3 C00081 BC00081  +REFP EC00081
CALL JOB:SEARCH-R1-S13D
SET P023 P006
SFTON3D P023
SMOVL C00082 BC00082 V=166.7  +MOVJ EC00082
MOVL C00083 BC00083 V=1000.0  +MOVJ EC00083 VJ=100.00
'EndPath S3401
MOVJ C00084 BC00084 VJ=100.00  +MOVJ EC00084 VJ=100.00
MOVJ C00085 BC00085 VJ=100.00  +MOVJ EC00085 VJ=100.00
'Path S3402
SFTOF3D
MOVJ C00086 BC00086 VJ=100.00  +MOVJ EC00086 VJ=100.00
MOVL C00087 BC00087 V=800.0  +MOVJ EC00087 VJ=100.00
SMOVL C00088 BC00088 V=166.7  +MOVJ EC00088
SREFP 3 C00089 BC00089  +REFP EC00089
CALL JOB:SEARCH-R1-S13D
SET P024 P006
SFTON3D P024
SMOVL C00090 BC00090 V=166.7  +MOVJ EC00090
SREFP 3 C00091 BC00091  +REFP EC00091
CALL JOB:SEARCH-R1-S13D
SET P024 P006
SFTON3D P024
SMOVL C00092 BC00092 V=250.0  +MOVJ EC00092
MOVL C00093 BC00093 V=1000.0  +MOVJ EC00093 VJ=100.00
'EndPath S3402
MOVJ C00094 BC00094 VJ=100.00  +MOVJ EC00094 VJ=100.00
MOVJ C00095 BC00095 VJ=100.00  +MOVJ EC00095 VJ=100.00
'Path S3403
SFTOF3D
MOVJ C00096 BC00096 VJ=100.00  +MOVJ EC00096 VJ=100.00
MOVL C00097 BC00097 V=800.0  +MOVJ EC00097 VJ=100.00
SMOVL C00098 BC00098 V=166.7  +MOVJ EC00098
SREFP 3 C00099 BC00099  +REFP EC00099
CALL JOB:SEARCH-R1-S13D
SET P025 P006
SFTON3D P025
SMOVL C00100 BC00100 V=166.7  +MOVJ EC00100
SREFP 3 C00101 BC00101  +REFP EC00101
CALL JOB:SEARCH-R1-S13D
SET P025 P006
SFTON3D P025
SMOVL C00102 BC00102 V=250.0  +MOVJ EC00102
MOVL C00103 BC00103 V=1000.0  +MOVJ EC00103 VJ=100.00
'EndPath S3403
MOVJ C00104 BC00104 VJ=100.00  +MOVJ EC00104 VJ=100.00
MOVJ C00105 BC00105 VJ=100.00  +MOVJ EC00105 VJ=100.00
'Path S3404
SFTOF3D
MOVJ C00106 BC00106 VJ=100.00  +MOVJ EC00106 VJ=100.00
MOVL C00107 BC00107 V=800.0  +MOVJ EC00107 VJ=100.00
SMOVL C00108 BC00108 V=166.7  +MOVJ EC00108
SREFP 3 C00109 BC00109  +REFP EC00109
CALL JOB:SEARCH-R1-S13D
SET P026 P006
SFTON3D P026
SMOVL C00110 BC00110 V=166.7  +MOVJ EC00110
SREFP 3 C00111 BC00111  +REFP EC00111
CALL JOB:SEARCH-R1-S13D
SET P026 P006
SFTON3D P026
SMOVL C00112 BC00112 V=166.7  +MOVJ EC00112
MOVL C00113 BC00113 V=1000.0  +MOVJ EC00113 VJ=100.00
'EndPath S3404
MOVJ C00114 BC00114 VJ=100.00  +MOVJ EC00114 VJ=100.00
MOVJ C00115 BC00115 VJ=100.00  +MOVJ EC00115 VJ=100.00
'
'
'
'Path W3405
SFTOF3D
SFTON3D P026
MOVJ C00116 BC00116 VJ=100.00  +MOVJ EC00116 VJ=100.00
SMOVL C00117 BC00117 V=800.0  +MOVJ EC00117
'POMINAC BO POSPAWANA
SMOVL C00118 BC00118 V=150.0 PL=0  +MOVJ EC00118
MACRO1 MJ#(0) ARGF21
ARCON
SWVON WEV#(108)
SMOVL C00119 BC00119 V=10.8  +MOVJ EC00119
SMOVL C00120 BC00120 V=10.8  +MOVJ EC00120
SMOVL C00121 BC00121 V=10.8  +MOVJ EC00121
ARCOF
SWVOF
SMOVL C00122 BC00122 V=800.0  +MOVJ EC00122
SMOVL C00123 BC00123 V=1000.0  +MOVJ EC00123
SFTOF3D
'EndPath W3405
MOVJ C00124 BC00124 VJ=100.00  +MOVJ EC00124 VJ=100.00
MOVJ C00125 BC00125 VJ=100.00  +MOVJ EC00125 VJ=100.00
'Path W3406
SFTOF3D
SFTON3D P021
MOVJ C00126 BC00126 VJ=100.00  +MOVJ EC00126 VJ=100.00
SMOVL C00127 BC00127 V=800.0  +MOVJ EC00127
SMOVL C00128 BC00128 V=150.0 PL=0  +MOVJ EC00128
MACRO1 MJ#(0) ARGF22
ARCON
SWVON WEV#(108)
SMOVL C00129 BC00129 V=10.8  +MOVJ EC00129
SMOVL C00130 BC00130 V=10.8  +MOVJ EC00130
SMOVL C00131 BC00131 V=10.8  +MOVJ EC00131
ARCOF
SWVOF
SMOVL C00132 BC00132 V=800.0  +MOVJ EC00132
SMOVL C00133 BC00133 V=1000.0  +MOVJ EC00133
SFTOF3D
'EndPath W3406
MOVJ C00134 BC00134 VJ=100.00  +MOVJ EC00134 VJ=100.00
MOVJ C00135 BC00135 VJ=100.00  +MOVJ EC00135 VJ=100.00
'Path W3407
SFTOF3D
SFTON3D P023
MOVJ C00136 BC00136 VJ=100.00  +MOVJ EC00136 VJ=100.00
SMOVL C00137 BC00137 V=800.0  +MOVJ EC00137
SMOVL C00138 BC00138 V=150.0 PL=0  +MOVJ EC00138
ARCON
SWVON WEV#(108)
SMOVL C00139 BC00139 V=10.8  +MOVJ EC00139
SMOVL C00140 BC00140 V=10.8  +MOVJ EC00140
SMOVL C00141 BC00141 V=10.8  +MOVJ EC00141
ARCOF
SWVOF
SMOVL C00142 BC00142 V=800.0  +MOVJ EC00142
SMOVL C00143 BC00143 V=1000.0  +MOVJ EC00143
SFTOF3D
'EndPath W3407
MOVJ C00144 BC00144 VJ=100.00  +MOVJ EC00144 VJ=100.00
MOVJ C00145 BC00145 VJ=100.00  +MOVJ EC00145 VJ=100.00
'Path W3408
SFTOF3D
SFTON3D P025
MOVJ C00146 BC00146 VJ=100.00  +MOVJ EC00146 VJ=100.00
SMOVL C00147 BC00147 V=800.0  +MOVJ EC00147
SMOVL C00148 BC00148 V=150.0 PL=0  +MOVJ EC00148
ARCON
SWVON WEV#(108)
SMOVL C00149 BC00149 V=10.8  +MOVJ EC00149
SMOVL C00150 BC00150 V=10.8  +MOVJ EC00150
SMOVL C00151 BC00151 V=10.8  +MOVJ EC00151
ARCOF
SWVOF
SMOVL C00152 BC00152 V=800.0  +MOVJ EC00152
SMOVL C00153 BC00153 V=1000.0  +MOVJ EC00153
SFTOF3D
'EndPath W3408
MOVJ C00154 BC00154 VJ=100.00  +MOVJ EC00154 VJ=100.00
MOVJ C00155 BC00155 VJ=100.00  +MOVJ EC00155 VJ=100.00
'Path W3409
SFTOF3D
SFTON3D P022
MOVJ C00156 BC00156 VJ=100.00  +MOVJ EC00156 VJ=100.00
SMOVL C00157 BC00157 V=800.0  +MOVJ EC00157
SMOVL C00158 BC00158 V=150.0 PL=0  +MOVJ EC00158
ARCON
SWVON WEV#(108)
SMOVL C00159 BC00159 V=10.8  +MOVJ EC00159
SMOVL C00160 BC00160 V=10.8  +MOVJ EC00160
SMOVL C00161 BC00161 V=10.8  +MOVJ EC00161
ARCOF
SWVOF
SMOVL C00162 BC00162 V=800.0  +MOVJ EC00162
SMOVL C00163 BC00163 V=1000.0  +MOVJ EC00163
SFTOF3D
'EndPath W3409
MOVJ C00164 BC00164 VJ=100.00  +MOVJ EC00164 VJ=100.00
MOVJ C00165 BC00165 VJ=100.00  +MOVJ EC00165 VJ=100.00
'Path W3410
SFTOF3D
SFTON3D P024
MOVJ C00166 BC00166 VJ=100.00  +MOVJ EC00166 VJ=100.00
SMOVL C00167 BC00167 V=800.0  +MOVJ EC00167
SMOVL C00168 BC00168 V=150.0 PL=0  +MOVJ EC00168
ARCON
SWVON WEV#(108)
SMOVL C00169 BC00169 V=10.8  +MOVJ EC00169
SMOVL C00170 BC00170 V=10.8  +MOVJ EC00170
SMOVL C00171 BC00171 V=10.8  +MOVJ EC00171
ARCOF
SWVOF
SMOVL C00172 BC00172 V=800.0  +MOVJ EC00172
SMOVL C00173 BC00173 V=1000.0  +MOVJ EC00173
SFTOF3D
'EndPath W3410
MOVJ C00174 BC00174 VJ=100.00  +MOVJ EC00174 VJ=100.00
'offset 20mm i synchro
MOVJ C00175 BC00175 VJ=100.00  +MOVJ EC00175 VJ=100.00
MOVJ C00176 BC00176 VJ=100.00  +MOVJ EC00176 VJ=100.00
'Path W3397
SFTOF3D
SFTON3D P027
MOVJ C00177 BC00177 VJ=100.00  +MOVJ EC00177 VJ=100.00
SMOVL C00178 BC00178 V=800.0  +MOVJ EC00178
REFP 1 RB1 C00179 BC00179
REFP 2 RB1 C00180 BC00180
SMOVL C00181 BC00181 V=150.0 PL=0  +MOVJ EC00179
ARCON
SWVON WEV#(100)
SMOVC C00182 BC00182 V=9.2  +MOVJ EC00180
SMOVC C00183 BC00183 V=9.2  +MOVJ EC00181
SMOVC C00184 BC00184 V=9.2  +MOVJ EC00182
SMOVC C00185 BC00185 V=9.2  +MOVJ EC00183
SFTON3D P066
SMOVL C00186 BC00186 V=9.2  +MOVJ EC00184
SMOVC C00187 BC00187 V=9.2  +MOVJ EC00185
SMOVC C00188 BC00188 V=9.2  +MOVJ EC00186
SMOVC C00189 BC00189 V=9.2  +MOVJ EC00187
SMOVL C00190 BC00190 V=9.2  +MOVJ EC00188
SMOVC C00191 BC00191 V=9.2  +MOVJ EC00189
SMOVC C00192 BC00192 V=9.2  +MOVJ EC00190
SFTON3D P067
SMOVC C00193 BC00193 V=9.2  +MOVJ EC00191
SMOVL C00194 BC00194 V=9.2  +MOVJ EC00192
SMOVC C00195 BC00195 V=9.2  +MOVJ EC00193
SMOVC C00196 BC00196 V=9.2  +MOVJ EC00194
SMOVC C00197 BC00197 V=9.2  +MOVJ EC00195
ARCOF
SWVOF
SMOVL C00198 BC00198 V=800.0  +MOVJ EC00196
SFTOF3D
SMOVL C00199 BC00199 V=1000.0  +MOVJ EC00197
SMOVL C00200 BC00200 V=1000.0  +MOVJ EC00198
SFTOF3D
'EndPath W3397
MOVJ C00201 BC00201 VJ=80.00  +MOVJ EC00199 VJ=80.00
'Path W3398
SFTOF3D
SFTON3D P028
MOVJ C00202 BC00202 VJ=100.00  +MOVJ EC00200 VJ=100.00
SMOVL C00203 BC00203 V=800.0  +MOVJ EC00201
REFP 1 RB1 C00204 BC00204
REFP 2 RB1 C00205 BC00205
SMOVL C00206 BC00206 V=166.7 PL=0  +MOVJ EC00202
ARCON
SWVON WEV#(100)
SMOVC C00207 BC00207 V=9.2  +MOVJ EC00203
SMOVC C00208 BC00208 V=9.2  +MOVJ EC00204
SMOVC C00209 BC00209 V=9.2  +MOVJ EC00205
SMOVC C00210 BC00210 V=9.2  +MOVJ EC00206
SMOVL C00211 BC00211 V=9.2  +MOVJ EC00207
SMOVC C00212 BC00212 V=9.2  +MOVJ EC00208
SMOVC C00213 BC00213 V=9.2  +MOVJ EC00209
SFTON3D P075
SMOVC C00214 BC00214 V=9.2  +MOVJ EC00210
SMOVC C00215 BC00215 V=9.2  +MOVJ EC00211
SMOVC C00216 BC00216 V=9.2  +MOVJ EC00212
SMOVC C00217 BC00217 V=9.2  +MOVJ EC00213
SFTON3D P068
SMOVC C00218 BC00218 V=9.2  +MOVJ EC00214
SMOVL C00219 BC00219 V=9.2  +MOVJ EC00215
SMOVC C00220 BC00220 V=9.2  +MOVJ EC00216
SMOVC C00221 BC00221 V=9.2  +MOVJ EC00217
SMOVC C00222 BC00222 V=9.2  +MOVJ EC00218
SMOVC C00223 BC00223 V=9.2  +MOVJ EC00219
ARCOF
SWVOF
SMOVL C00224 BC00224 V=800.0  +MOVJ EC00220
SMOVL C00225 BC00225 V=1000.0  +MOVJ EC00221
SMOVL C00226 BC00226 V=1000.0  +MOVJ EC00222
SFTOF3D
MOVJ C00227 BC00227 VJ=50.00  +MOVJ EC00223 VJ=50.00
'EndPath W3398
MOVJ C00228 BC00228 VJ=50.00  +MOVJ EC00224 VJ=100.00
MOVJ C00229 BC00229 VJ=50.00  +MOVJ EC00225 VJ=100.00
END
